FUNCTION FUN_InsideHysteresis360 : BOOL
VAR_INPUT
	rAct		:REAL;			// Actual value
	rSp			:REAL;			// Setpoint value
	rHys		:REAL;			// Hysteresis	
END_VAR
VAR
	bInside		:BOOL;			// True if actual value is within setpoint plus minus hysteresis value
END_VAR



// Determine if value is close to loop back point at 360 Deg. 
IF (rSp+rHys) > 360.0000 OR (rSp-rHys) < 0.0000 THEN
	// SP is close to switch
	IF (rSp+rHys) > 360.0000 THEN
		// High limit is above 360 deg
		IF (rAct >= (rSp-rHys)) OR (rAct <= (rSp+rHys-360)) THEN
 			bInside := TRUE;
		ELSE
			bInside := FALSE;
		END_IF
	ELSE 
		IF (rAct <= (rSp+rHys)) OR (rAct >= (360+(rSP-rHys))) THEN 
			bInside := TRUE;
		ELSE
			bInside := FALSE;
		END_IF
	END_IF
ELSE
	// SP is not close to 0 or 360 deg.
	bInside := FUN_InsideHysteresis(rAct:= rAct, rSp:= rSp, rHys:= rHys);
END_IF

// Set return value
FUN_InsideHysteresis360 := bInside;

END_FUNCTION

(* stored: Version 1.1.0.1, ProductVersion 3.1.4024.12
   POU FUN_InsideHysteresis360: Id {87050e55-6a88-4571-b4a1-ec1f003085b4}, SpecialFunc None *)
